// TIA Portal project "FactoryIO_Template_S7-1200_V15_V18" (V18)
// Vorlageprojekt für das Buch mit Zielsystem S7-1200

(* hardware
DEVICE "S7-1200-Station_1"  S7-1200 Station
   slot 0: "Baugruppenträger_0"  Rack  V1.0
   slot 1: "PLC_1"  CPU 1211C DC/DC/DC  6ES7 211-1AE40-0XB0  V4.1
DEVICE "HMI_1"  TP700 Comfort
   slot 0: "HMI_1"  TP700 Comfort  6AV2 124-0GC01-0AX0  17.0.0.0
   slot 1: "HMI_RT_1"  TP700 Comfort  6AV2 124-0GC01-0AX0  17.0.0.0
   slot 5: "HMI_1.IE_CP_1"  PROFINET Interface  17.0.0.0
      slot 1: "PROFINET Interface_1"  PROFINET Interface
         slot 1: "Port_1"  Port
         slot 2: "Port_2"  Port
   slot 7: "HMI_1.MPI/DP_CP_1"  MPI/DP Interface  17.0.0.0
DEVICE "PC station"  SIMATIC PC station
   slot 0: "PC station"  Rail  SIMATIC PC-Station  V1.0
      slot 125: "Stationmanager"  Station_Manager  V6.0.4
   slot 1: "IE general_1"  IE General  IE_CP  V8.2.0
      slot 1: "PROFINET interface"  IEGeneral.Interface.8.2.0
   slot 2: "HMI_RT_2"  WinCC RT Advanced  6AV2 104-0xxxx-xxxx  17.0.0.0
      slot 33792: "Computer interface"  Host interface
*)

// ===== PLC "PLC_1"  CPU 1211C DC/DC/DC =====

VAR_GLOBAL   // PLC tag table "Standard-Variablentabelle"
   "item at inter 0" AT %I0.0 : Bool;
   "item at exit 0" AT %I0.1 : Bool;
   "moving x0" AT %I0.2 : Bool;
   "moving z0" AT %I0.3 : Bool;
   "item detect 0" AT %I0.4 : Bool;
   "Start Button 0" AT %I0.5 : Bool;
   "Stop Button 0" AT %I0.6 : Bool;
   "Emergency Stop 0" AT %I0.7 : Bool;
   "enter conveyor (4m) 0" AT %Q0.0 : Bool;
   "exit conveyor (4m) 0" AT %Q0.1 : Bool;
   "move x0" AT %Q0.2 : Bool;
   "move z0" AT %Q0.3 : Bool;
   "grab 0" AT %Q0.4 : Bool;
   "Start Button 0 (Light)" AT %Q0.5 : Bool;
   "Stop Button 0 (Light)" AT %Q0.6 : Bool;
   "State0" AT %M1.0 : Bool;
   "State1" AT %M1.1 : Bool;
   "State2" AT %M1.2 : Bool;
   "State3" AT %M1.3 : Bool;
   "State4" AT %M1.4 : Bool;
   "State5" AT %M1.5 : Bool;
   "State6" AT %M1.6 : Bool;
   "State7" AT %M1.7 : Bool;
   "State8" AT %M2.0 : Bool;
   "State9" AT %M2.1 : Bool;
   "Tag_1" AT %M2.2 : Bool;
   "Tag_2" AT %M0.3 : Bool;
   "Tag_3" AT %M0.4 : Bool;
   "Tag_4" AT %M0.5 : Bool;
   "Tag_5" AT %M0.6 : Bool;
   "Tag_6" AT %M0.7 : Bool;
   "Digital Display 0" AT %QD30 : DInt;
   "Belt Conveyor (2m) 0" AT %Q0.7 : Bool;
   "Reset Button 0" AT %I1.0 : Bool;
   "Pusher 0" AT %Q1.0 : Bool;
   "Tag_7" AT %M0.0 : Bool;
   "Vision Sensor 3" AT %I1.1 : Bool;
   "Belt Conveyor (6m) 0" AT %Q1.1 : Bool;
   "Belt Conveyor (6m) 1" AT %Q1.2 : Bool;
   "Curved Belt Conveyor 0 CCW" AT %Q1.3 : Bool;
   "Curved Belt Conveyor 1 CW" AT %Q1.4 : Bool;
   "Belt Conveyor (6m) 2c1" AT %Q1.5 : Bool;
   "Belt Conveyor (6m) c_3_1" AT %Q1.6 : Bool;
   "Enter_sensor_green1" AT %I1.2 : Bool;
   "Exit_sensor_green" AT %I1.3 : Bool;
   "pusher_sensor" AT %I1.4 : Bool;
   "pusher_Sensor 2" AT %I1.5 : Bool;
   "Belt Conveyor (6m) 4" AT %Q1.7 : Bool;
   "Belt Conveyor (6m) 5" AT %Q2.0 : Bool;
   "Machining green(Start)" AT %Q2.1 : Bool;
   "Machining green  (Stop)" AT %Q2.2 : Bool;
   "Belt Conveyor (4m) 2c2" AT %Q2.3 : Bool;
   "Tag_8" AT %M2.3 : Bool;
   "reset_c1" AT %M2.4 : Bool;
   "Tag_9" AT %M2.5 : Bool;
   "Tag_10" AT %MW200 : Word;
   "reset_marker_lids" AT %M2.6 : Bool;
   "Tag_11" AT %M2.7 : Bool;
   "reset_c_1_b" AT %M3.0 : Bool;
   "Tag_12" AT %M3.1 : Bool;
   "reset_lib_blue" AT %M3.2 : Bool;
   "Tag_14" AT %MW300 : Int;
   "Tag_13" AT %M3.3 : Bool;
   "Tag_15" AT %M3.4 : Bool;
   "Tag_16" AT %M3.5 : Bool;
   "Tag_17" AT %M3.6 : Bool;
   "Tag_18" AT %M3.7 : Bool;
   "Tag_19" AT %M4.0 : Bool;
   "Tag_20" AT %M4.1 : Bool;
   "Tag_21" AT %M4.2 : Bool;
   "Tag_22" AT %M4.3 : Bool;
   "Tag_23" AT %M4.4 : Bool;
   "Tag_24" AT %M4.5 : Bool;
   "Tag_25" AT %M4.6 : Bool;
   "Tag_26" AT %M5.0 : Bool;
   "Tag_27" AT %M5.1 : Bool;
   "Tag_28" AT %M5.2 : Bool;
   "Tag_29" AT %M5.3 : Bool;
   "Tag_30" AT %M5.4 : Bool;
   "Tag_31" AT %MW400 : Int;
   "Tag_32" AT %M5.5 : Bool;
   "Tag_33" AT %MW500 : Int;
   "Tag_34" AT %MW600 : Int;
   "Tag_35" AT %M5.6 : Bool;
END_VAR

VAR_GLOBAL   // PLC tag table "Tag table from XML_1"
   "Digital Display 1" AT %QD34 : DInt;
   "Digital Display 2" AT %QD38 : DInt;
END_VAR

VAR_GLOBAL   // PLC tag table "Tag table from XML_4"
   "Enter_sensor_green2" AT %I1.6 : Bool;
END_VAR

VAR_GLOBAL   // PLC tag table "Tag table from XML_5"
   "Entry_sensor_blue_2_1" AT %I1.7 : Bool;
   "Entry_sensor_blue_2_2" AT %I2.0 : Bool;
   "Exit_sensor_blue_2" AT %I2.1 : Bool;
   "Start Button 1" AT %I2.2 : Bool;
   "Stop Button 1" AT %I2.3 : Bool;
   "Emergency Stop 1" AT %I2.4 : Bool;
   "Start Button 2" AT %I2.5 : Bool;
   "Stop Button 2" AT %I2.6 : Bool;
   "Emergency Stop 2" AT %I2.7 : Bool;
   "Start Button 3" AT %I3.0 : Bool;
   "Stop Button 3" AT %I3.1 : Bool;
   "Start Button 4" AT %I3.2 : Bool;
   "Stop Button 4" AT %I3.3 : Bool;
   "Moving X1" AT %I3.4 : Bool;
   "Moving Z1" AT %I3.5 : Bool;
   "Detected_item_1" AT %I3.6 : Bool;
   "Right Positioner 0 (Clamped)" AT %I3.7 : Bool;
   "Right Positioner 1 (Clamped)" AT %I4.0 : Bool;
   "Vision Sensor 0" AT %I4.1 : Bool;
   "Vision Sensor 1" AT %I4.2 : Bool;
   "push_sensor_2_1" AT %I4.3 : Bool;
   "push_sensor_2_2" AT %I4.4 : Bool;
   "push_sensor_3_1" AT %I4.5 : Bool;
   "push_sensor_3_2" AT %I4.6 : Bool;
   "counter_blue" AT %I4.7 : Bool;
   "counter_green" AT %I5.0 : Bool;
   "part_leveing1" AT %I5.1 : Bool;
   "part_leveing2" AT %I5.2 : Bool;
   "Moving X2" AT %I5.3 : Bool;
   "Moving Z2" AT %I5.4 : Bool;
   "Detected_item_2" AT %I5.5 : Bool;
   "Right Positioner 3 (Clamped)" AT %I5.6 : Bool;
   "Right Positioner 2 (Clamped)" AT %I5.7 : Bool;
   "Right Positioner 1 (Limit)" AT %I6.0 : Bool;
   "Right Positioner 3 (Limit)" AT %I6.1 : Bool;
   "Machining green lids" AT %Q2.4 : Bool;
   "Machining Center 0 (Produce Lids)" AT %Q2.5 : Bool;
   "Belt Conveyor (4m) c_3_2" AT %Q2.6 : Bool;
   "Start Button 1 (Light)" AT %Q2.7 : Bool;
   "Stop Button 1 (Light)" AT %Q3.0 : Bool;
   "Start Button 2 (Light)" AT %Q3.1 : Bool;
   "Stop Button 2 (Light)" AT %Q3.2 : Bool;
   "Start Button 3 (Light)" AT %Q3.3 : Bool;
   "Stop Button 3 (Light)" AT %Q3.4 : Bool;
   "Start Button 4 (Light)" AT %Q3.5 : Bool;
   "Stop Button 4 (Light)" AT %Q3.6 : Bool;
   "Curved Belt Conveyor 2 CCW" AT %Q3.7 : Bool;
   "Curved Belt Conveyor 3 CCW" AT %Q4.0 : Bool;
   "Belt Conveyor (4m) 3" AT %Q4.1 : Bool;
   "Belt Conveyor (4m) 4" AT %Q4.2 : Bool;
   "Belt Conveyor (4m) 5" AT %Q4.3 : Bool;
   "Belt Conveyor (4m) 6" AT %Q4.4 : Bool;
   "Move x1" AT %Q4.5 : Bool;
   "move z1" AT %Q4.6 : Bool;
   "Pusher _2" AT %Q4.7 : Bool;
   "Right Positioner 0 (Clamp)" AT %Q5.0 : Bool;
   "Right Positioner 1 (Clamp)" AT %Q5.1 : Bool;
   "Pusher_3" AT %Q5.2 : Bool;
   "Belt Conveyor (4m) 8" AT %Q5.3 : Bool;
   "Belt Conveyor (4m) 9" AT %Q5.4 : Bool;
   "Belt Conveyor (4m) 10" AT %Q5.5 : Bool;
   "Belt Conveyor (4m) 11" AT %Q5.6 : Bool;
   "move X2" AT %Q5.7 : Bool;
   "move z2" AT %Q6.0 : Bool;
   "Grab2" AT %Q6.1 : Bool;
   "Right Positioner 3 (Clamp)" AT %Q6.2 : Bool;
   "Right Positioner 2 (Clamp)" AT %Q6.3 : Bool;
   "Right Positioner 1 (Raise)" AT %Q6.4 : Bool;
   "Right Positioner 3 (Raise)" AT %Q6.5 : Bool;
END_VAR

VAR_GLOBAL   // PLC tag table "Tag table from XML_6"
   "Machining blue 0 (Start)" AT %Q6.6 : Bool;
   "Machining blue 0 (Stop)" AT %Q6.7 : Bool;
END_VAR

VAR_GLOBAL   // PLC tag table "Tag table from XML_7"
   "Grab1" AT %Q7.0 : Bool;
END_VAR

VAR_GLOBAL   // PLC tag table "Tag table from XML_8"
   "lid_place_blue" AT %I6.2 : Bool;
   "base_place_blue" AT %I6.3 : Bool;
   "lid_place_green" AT %I6.4 : Bool;
   "base_place_green" AT %I6.5 : Bool;
END_VAR

// folder: System blocks/Program resources

DATA_BLOCK "IEC_Counter_0_DB"   // DB1
{ S7_Optimized_Access := 'TRUE' }
AUTHOR : Simatic
FAMILY : IEC
NAME : CNTR
VERSION : 1.0
// stored: InstanceOfName IEC_COUNTER
"IEC_COUNTER"
BEGIN
END_DATA_BLOCK

DATA_BLOCK "IEC_Timer_0_DB"   // DB2
{ S7_Optimized_Access := 'TRUE' }
AUTHOR : Simatic
FAMILY : IEC
NAME : IEC_TMR
VERSION : 1.0
// stored: InstanceOfName IEC_TIMER
"IEC_TIMER"
BEGIN
END_DATA_BLOCK

DATA_BLOCK "IEC_Timer_0_DB_1"   // DB3
{ S7_Optimized_Access := 'TRUE' }
AUTHOR : Simatic
FAMILY : IEC
NAME : IEC_TMR
VERSION : 1.0
// stored: InstanceOfName IEC_TIMER
"IEC_TIMER"
BEGIN
END_DATA_BLOCK

DATA_BLOCK "produce_lids_counter"   // DB4
{ S7_Optimized_Access := 'TRUE' }
AUTHOR : Simatic
FAMILY : IEC
NAME : CNTR
VERSION : 1.0
// stored: InstanceOfName IEC_COUNTER
"IEC_COUNTER"
BEGIN
END_DATA_BLOCK

DATA_BLOCK "IEC_Timer_0_DB_2"   // DB5
{ S7_Optimized_Access := 'TRUE' }
AUTHOR : Simatic
FAMILY : IEC
NAME : IEC_TMR
VERSION : 1.0
// stored: InstanceOfName IEC_TIMER
"IEC_TIMER"
BEGIN
END_DATA_BLOCK

DATA_BLOCK "IEC_Timer_0_DB_3"   // DB6
{ S7_Optimized_Access := 'TRUE' }
AUTHOR : Simatic
FAMILY : IEC
NAME : IEC_TMR
VERSION : 1.0
// stored: InstanceOfName IEC_TIMER
"IEC_TIMER"
BEGIN
END_DATA_BLOCK

DATA_BLOCK "produce_lids_counter_blue"   // DB7
{ S7_Optimized_Access := 'TRUE' }
AUTHOR : Simatic
FAMILY : IEC
NAME : CNTR
VERSION : 1.0
// stored: InstanceOfName IEC_COUNTER
"IEC_COUNTER"
BEGIN
END_DATA_BLOCK

DATA_BLOCK "Green_Product_Counter"   // DB9
{ S7_Optimized_Access := 'TRUE' }
AUTHOR : Simatic
FAMILY : IEC
NAME : CNTR
VERSION : 1.0
// stored: InstanceOfName IEC_COUNTER
"IEC_COUNTER"
BEGIN
END_DATA_BLOCK

DATA_BLOCK "Blue_Product_Counter"   // DB10
{ S7_Optimized_Access := 'TRUE' }
AUTHOR : Simatic
FAMILY : IEC
NAME : CNTR
VERSION : 1.0
// stored: InstanceOfName IEC_COUNTER
"IEC_COUNTER"
BEGIN
END_DATA_BLOCK

// folder: (top level)

FUNCTION "Start_Stop" : Void   // FC1, LAD
{ S7_Optimized_Access := 'TRUE' }
VERSION : 0.1
BEGIN

REGION Network 1
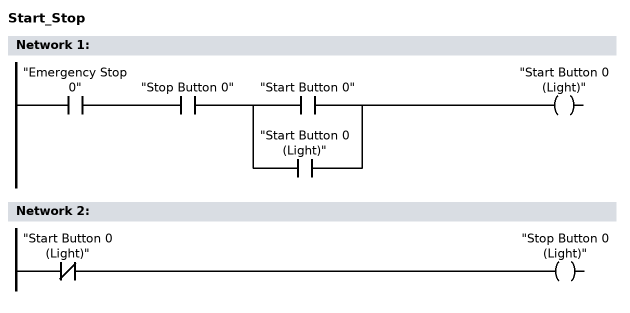
   RUNG wire#powerrail
      Contact( "Emergency Stop 0" )
      Contact( "Stop Button 0" )
      wire#w1
      Contact( "Start Button 0" )
      wire#w2
      Coil( "Start Button 0 (Light)" )
   END_RUNG
   RUNG wire#w1
      Contact( "Start Button 0 (Light)" )
   END_RUNG wire#w2
   // the same network as SCL:
   "Start Button 0 (Light)" := "Emergency Stop 0" AND "Stop Button 0" AND ("Start Button 0" OR "Start Button 0 (Light)");
END_REGION

REGION Network 2
   RUNG wire#powerrail
      I_Contact( "Start Button 0 (Light)" )
      Coil( "Stop Button 0 (Light)" )
   END_RUNG
   // the same network as SCL:
   "Stop Button 0 (Light)" := NOT "Start Button 0 (Light)";
END_REGION
END_FUNCTION

FUNCTION "States" : Void   // FC2, LAD
{ S7_Optimized_Access := 'TRUE' }
VERSION : 0.1
   VAR_TEMP   // added for the SCL form of the ladder/FBD networks
      _w1 : Bool;
   END_VAR
BEGIN

REGION Network 1: State0
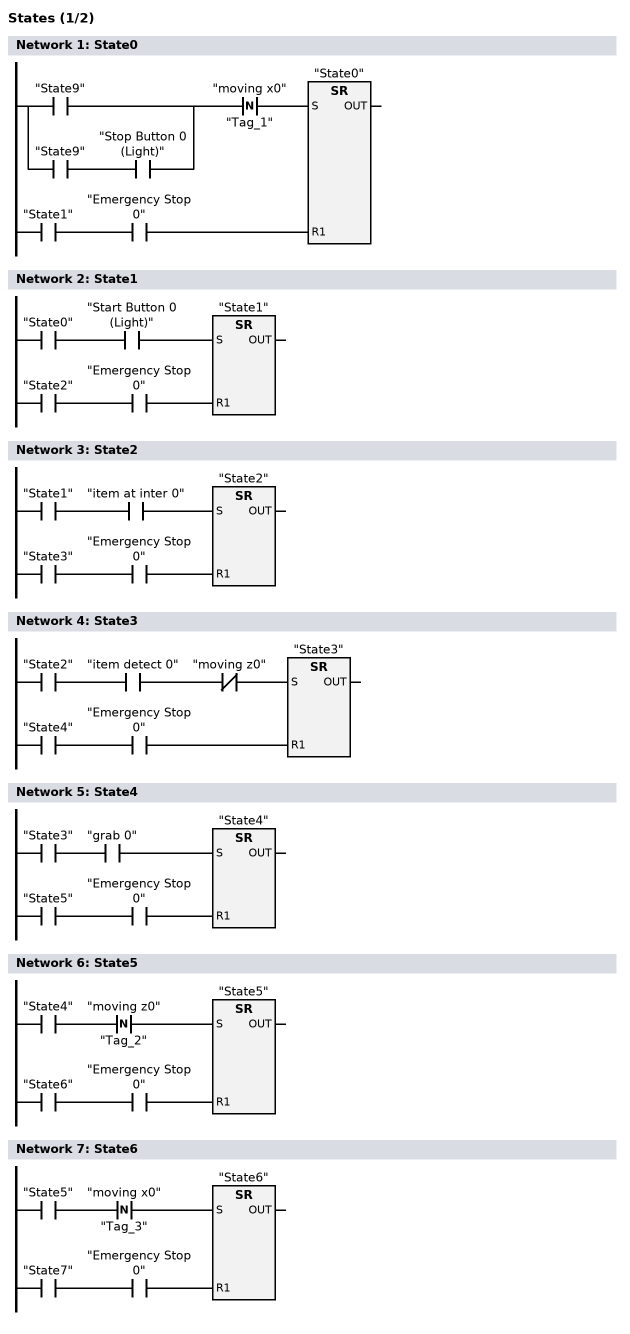
   RUNG wire#powerrail
      Contact( "State9" )
      wire#w1
      N_Contact(operand := "moving x0", bit := "Tag_1")
      S_SR(operand := "State0", r1 := wire#w2)
   END_RUNG
   RUNG wire#powerrail
      Contact( "State9" )
      Contact( "Stop Button 0 (Light)" )
   END_RUNG wire#w1
   RUNG wire#powerrail
      Contact( "State1" )
      Contact( "Emergency Stop 0" )
   END_RUNG wire#w2
   // the same network as SCL:
   #_w1 := ("State9" OR ("State9" AND "Stop Button 0 (Light)")) AND NOT "moving x0" AND "Tag_1";   // falling edge of "moving x0"
   "Tag_1" := "moving x0";
   IF #_w1 THEN
       "State0" := TRUE;   // SR flip-flop
   END_IF;
   IF "State1" AND "Emergency Stop 0" THEN "State0" := FALSE; END_IF;
END_REGION

REGION Network 2: State1
   RUNG wire#powerrail
      Contact( "State0" )
      Contact( "Start Button 0 (Light)" )
      S_SR(operand := "State1", r1 := wire#w1)
   END_RUNG
   RUNG wire#powerrail
      Contact( "State2" )
      Contact( "Emergency Stop 0" )
   END_RUNG wire#w1
   // the same network as SCL:
   IF "State0" AND "Start Button 0 (Light)" THEN
       "State1" := TRUE;   // SR flip-flop
   END_IF;
   IF "State2" AND "Emergency Stop 0" THEN "State1" := FALSE; END_IF;
END_REGION

REGION Network 3: State2
   RUNG wire#powerrail
      Contact( "State1" )
      Contact( "item at inter 0" )
      S_SR(operand := "State2", r1 := wire#w1)
   END_RUNG
   RUNG wire#powerrail
      Contact( "State3" )
      Contact( "Emergency Stop 0" )
   END_RUNG wire#w1
   // the same network as SCL:
   IF "State1" AND "item at inter 0" THEN
       "State2" := TRUE;   // SR flip-flop
   END_IF;
   IF "State3" AND "Emergency Stop 0" THEN "State2" := FALSE; END_IF;
END_REGION

REGION Network 4: State3
   RUNG wire#powerrail
      Contact( "State2" )
      Contact( "item detect 0" )
      I_Contact( "moving z0" )
      S_SR(operand := "State3", r1 := wire#w1)
   END_RUNG
   RUNG wire#powerrail
      Contact( "State4" )
      Contact( "Emergency Stop 0" )
   END_RUNG wire#w1
   // the same network as SCL:
   IF "State2" AND "item detect 0" AND NOT "moving z0" THEN
       "State3" := TRUE;   // SR flip-flop
   END_IF;
   IF "State4" AND "Emergency Stop 0" THEN "State3" := FALSE; END_IF;
END_REGION

REGION Network 5: State4
   RUNG wire#powerrail
      Contact( "State3" )
      Contact( "grab 0" )
      S_SR(operand := "State4", r1 := wire#w1)
   END_RUNG
   RUNG wire#powerrail
      Contact( "State5" )
      Contact( "Emergency Stop 0" )
   END_RUNG wire#w1
   // the same network as SCL:
   IF "State3" AND "grab 0" THEN
       "State4" := TRUE;   // SR flip-flop
   END_IF;
   IF "State5" AND "Emergency Stop 0" THEN "State4" := FALSE; END_IF;
END_REGION

REGION Network 6: State5
   RUNG wire#powerrail
      Contact( "State4" )
      N_Contact(operand := "moving z0", bit := "Tag_2")
      S_SR(operand := "State5", r1 := wire#w1)
   END_RUNG
   RUNG wire#powerrail
      Contact( "State6" )
      Contact( "Emergency Stop 0" )
   END_RUNG wire#w1
   // the same network as SCL:
   #_w1 := "State4" AND NOT "moving z0" AND "Tag_2";   // falling edge of "moving z0"
   "Tag_2" := "moving z0";
   IF #_w1 THEN
       "State5" := TRUE;   // SR flip-flop
   END_IF;
   IF "State6" AND "Emergency Stop 0" THEN "State5" := FALSE; END_IF;
END_REGION

REGION Network 7: State6
   RUNG wire#powerrail
      Contact( "State5" )
      N_Contact(operand := "moving x0", bit := "Tag_3")
      S_SR(operand := "State6", r1 := wire#w1)
   END_RUNG
   RUNG wire#powerrail
      Contact( "State7" )
      Contact( "Emergency Stop 0" )
   END_RUNG wire#w1
   // the same network as SCL:
   #_w1 := "State5" AND NOT "moving x0" AND "Tag_3";   // falling edge of "moving x0"
   "Tag_3" := "moving x0";
   IF #_w1 THEN
       "State6" := TRUE;   // SR flip-flop
   END_IF;
   IF "State7" AND "Emergency Stop 0" THEN "State6" := FALSE; END_IF;
END_REGION

REGION Network 8: State7
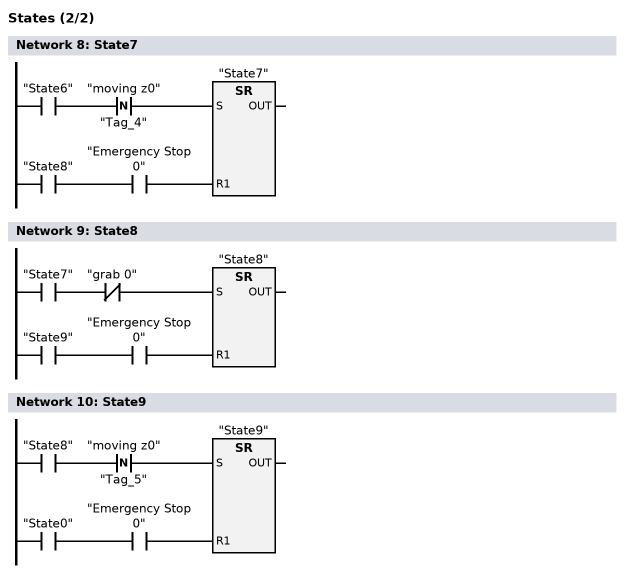
   RUNG wire#powerrail
      Contact( "State6" )
      N_Contact(operand := "moving z0", bit := "Tag_4")
      S_SR(operand := "State7", r1 := wire#w1)
   END_RUNG
   RUNG wire#powerrail
      Contact( "State8" )
      Contact( "Emergency Stop 0" )
   END_RUNG wire#w1
   // the same network as SCL:
   #_w1 := "State6" AND NOT "moving z0" AND "Tag_4";   // falling edge of "moving z0"
   "Tag_4" := "moving z0";
   IF #_w1 THEN
       "State7" := TRUE;   // SR flip-flop
   END_IF;
   IF "State8" AND "Emergency Stop 0" THEN "State7" := FALSE; END_IF;
END_REGION

REGION Network 9: State8
   RUNG wire#powerrail
      Contact( "State7" )
      I_Contact( "grab 0" )
      S_SR(operand := "State8", r1 := wire#w1)
   END_RUNG
   RUNG wire#powerrail
      Contact( "State9" )
      Contact( "Emergency Stop 0" )
   END_RUNG wire#w1
   // the same network as SCL:
   IF "State7" AND NOT "grab 0" THEN
       "State8" := TRUE;   // SR flip-flop
   END_IF;
   IF "State9" AND "Emergency Stop 0" THEN "State8" := FALSE; END_IF;
END_REGION

REGION Network 10: State9
   RUNG wire#powerrail
      Contact( "State8" )
      N_Contact(operand := "moving z0", bit := "Tag_5")
      S_SR(operand := "State9", r1 := wire#w1)
   END_RUNG
   RUNG wire#powerrail
      Contact( "State0" )
      Contact( "Emergency Stop 0" )
   END_RUNG wire#w1
   // the same network as SCL:
   #_w1 := "State8" AND NOT "moving z0" AND "Tag_5";   // falling edge of "moving z0"
   "Tag_5" := "moving z0";
   IF #_w1 THEN
       "State9" := TRUE;   // SR flip-flop
   END_IF;
   IF "State0" AND "Emergency Stop 0" THEN "State9" := FALSE; END_IF;
END_REGION
END_FUNCTION

FUNCTION "Actuators" : Void   // FC3, LAD
{ S7_Optimized_Access := 'TRUE' }
VERSION : 0.1
BEGIN

REGION Network 1
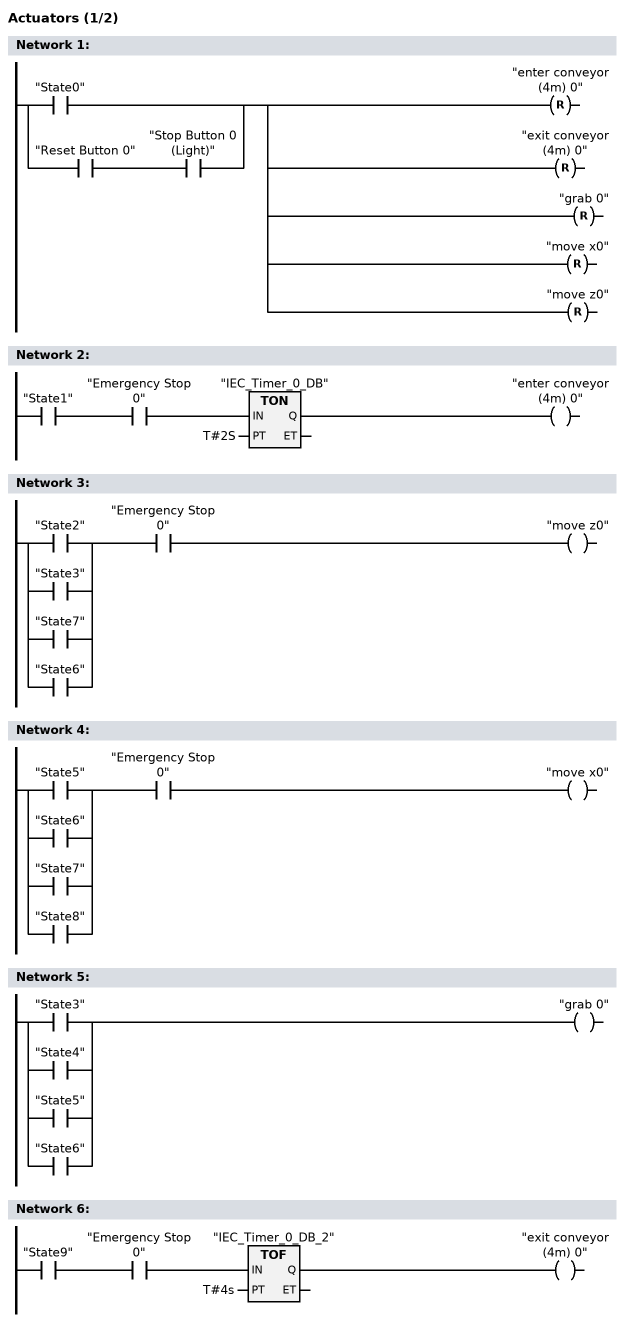
   RUNG wire#powerrail
      Contact( "State0" )
      wire#w1
      R_Coil( "enter conveyor (4m) 0" )
   END_RUNG
   RUNG wire#powerrail
      Contact( "Reset Button 0" )
      Contact( "Stop Button 0 (Light)" )
   END_RUNG wire#w1
   RUNG wire#w1
      R_Coil( "exit conveyor (4m) 0" )
   END_RUNG
   RUNG wire#w1
      R_Coil( "grab 0" )
   END_RUNG
   RUNG wire#w1
      R_Coil( "move x0" )
   END_RUNG
   RUNG wire#w1
      R_Coil( "move z0" )
   END_RUNG
   // the same network as SCL:
   IF "State0" OR ("Reset Button 0" AND "Stop Button 0 (Light)") THEN
       "enter conveyor (4m) 0" := FALSE;
       "exit conveyor (4m) 0" := FALSE;
       "grab 0" := FALSE;
       "move x0" := FALSE;
       "move z0" := FALSE;
   END_IF;
END_REGION

REGION Network 2
   "IEC_Timer_0_DB".TON(IN := "State1" AND "Emergency Stop 0", PT := T#2S);
   "enter conveyor (4m) 0" := "IEC_Timer_0_DB".Q;
END_REGION

REGION Network 3
   RUNG wire#powerrail
      Contact( "State2" )
      wire#w1
      Contact( "Emergency Stop 0" )
      Coil( "move z0" )
   END_RUNG
   RUNG wire#powerrail
      Contact( "State3" )
   END_RUNG wire#w1
   RUNG wire#powerrail
      Contact( "State7" )
   END_RUNG wire#w1
   RUNG wire#powerrail
      Contact( "State6" )
   END_RUNG wire#w1
   // the same network as SCL:
   "move z0" := ("State2" OR "State3" OR "State7" OR "State6") AND "Emergency Stop 0";
END_REGION

REGION Network 4
   RUNG wire#powerrail
      Contact( "State5" )
      wire#w1
      Contact( "Emergency Stop 0" )
      Coil( "move x0" )
   END_RUNG
   RUNG wire#powerrail
      Contact( "State6" )
   END_RUNG wire#w1
   RUNG wire#powerrail
      Contact( "State7" )
   END_RUNG wire#w1
   RUNG wire#powerrail
      Contact( "State8" )
   END_RUNG wire#w1
   // the same network as SCL:
   "move x0" := ("State5" OR "State6" OR "State7" OR "State8") AND "Emergency Stop 0";
END_REGION

REGION Network 5
   RUNG wire#powerrail
      Contact( "State3" )
      wire#w1
      Coil( "grab 0" )
   END_RUNG
   RUNG wire#powerrail
      Contact( "State4" )
   END_RUNG wire#w1
   RUNG wire#powerrail
      Contact( "State5" )
   END_RUNG wire#w1
   RUNG wire#powerrail
      Contact( "State6" )
   END_RUNG wire#w1
   // the same network as SCL:
   "grab 0" := "State3" OR "State4" OR "State5" OR "State6";
END_REGION

REGION Network 6
   "IEC_Timer_0_DB_2".TOF(IN := "State9" AND "Emergency Stop 0", PT := T#4s);
   "exit conveyor (4m) 0" := "IEC_Timer_0_DB_2".Q;
END_REGION

REGION Network 7
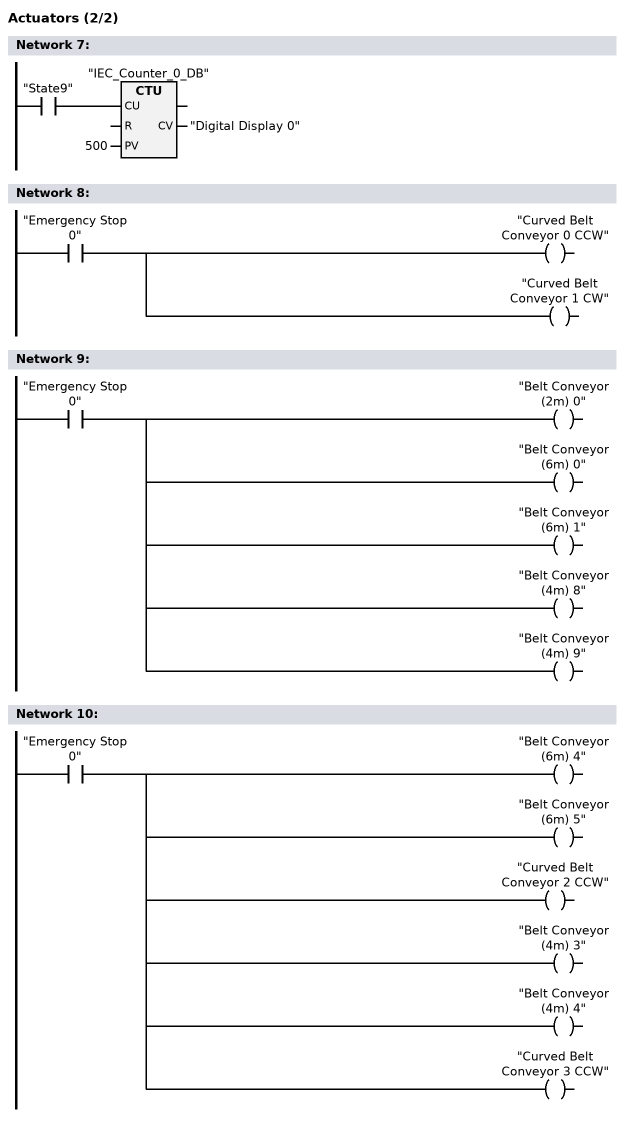
   "IEC_Counter_0_DB".CTU(CU := "State9", PV := 500, CV => "Digital Display 0");
END_REGION

REGION Network 8
   RUNG wire#powerrail
      Contact( "Emergency Stop 0" )
      wire#w1
      Coil( "Curved Belt Conveyor 0 CCW" )
   END_RUNG
   RUNG wire#w1
      Coil( "Curved Belt Conveyor 1 CW" )
   END_RUNG
   // the same network as SCL:
   "Curved Belt Conveyor 0 CCW" := "Emergency Stop 0";
   "Curved Belt Conveyor 1 CW" := "Emergency Stop 0";
END_REGION

REGION Network 9
   RUNG wire#powerrail
      Contact( "Emergency Stop 0" )
      wire#w1
      Coil( "Belt Conveyor (2m) 0" )
   END_RUNG
   RUNG wire#w1
      Coil( "Belt Conveyor (6m) 0" )
   END_RUNG
   RUNG wire#w1
      Coil( "Belt Conveyor (6m) 1" )
   END_RUNG
   RUNG wire#w1
      Coil( "Belt Conveyor (4m) 8" )
   END_RUNG
   RUNG wire#w1
      Coil( "Belt Conveyor (4m) 9" )
   END_RUNG
   // the same network as SCL:
   "Belt Conveyor (2m) 0" := "Emergency Stop 0";
   "Belt Conveyor (6m) 0" := "Emergency Stop 0";
   "Belt Conveyor (6m) 1" := "Emergency Stop 0";
   "Belt Conveyor (4m) 8" := "Emergency Stop 0";
   "Belt Conveyor (4m) 9" := "Emergency Stop 0";
END_REGION

REGION Network 10
   RUNG wire#powerrail
      Contact( "Emergency Stop 0" )
      wire#w1
      Coil( "Belt Conveyor (6m) 4" )
   END_RUNG
   RUNG wire#w1
      Coil( "Belt Conveyor (6m) 5" )
   END_RUNG
   RUNG wire#w1
      Coil( "Curved Belt Conveyor 2 CCW" )
   END_RUNG
   RUNG wire#w1
      Coil( "Belt Conveyor (4m) 3" )
   END_RUNG
   RUNG wire#w1
      Coil( "Belt Conveyor (4m) 4" )
   END_RUNG
   RUNG wire#w1
      Coil( "Curved Belt Conveyor 3 CCW" )
   END_RUNG
   // the same network as SCL:
   "Belt Conveyor (6m) 4" := "Emergency Stop 0";
   "Belt Conveyor (6m) 5" := "Emergency Stop 0";
   "Curved Belt Conveyor 2 CCW" := "Emergency Stop 0";
   "Belt Conveyor (4m) 3" := "Emergency Stop 0";
   "Belt Conveyor (4m) 4" := "Emergency Stop 0";
   "Curved Belt Conveyor 3 CCW" := "Emergency Stop 0";
END_REGION
END_FUNCTION

FUNCTION "CNC_BLUE" : Void   // FC4, LAD
{ S7_Optimized_Access := 'TRUE' }
VERSION : 0.1
BEGIN

REGION Network 1
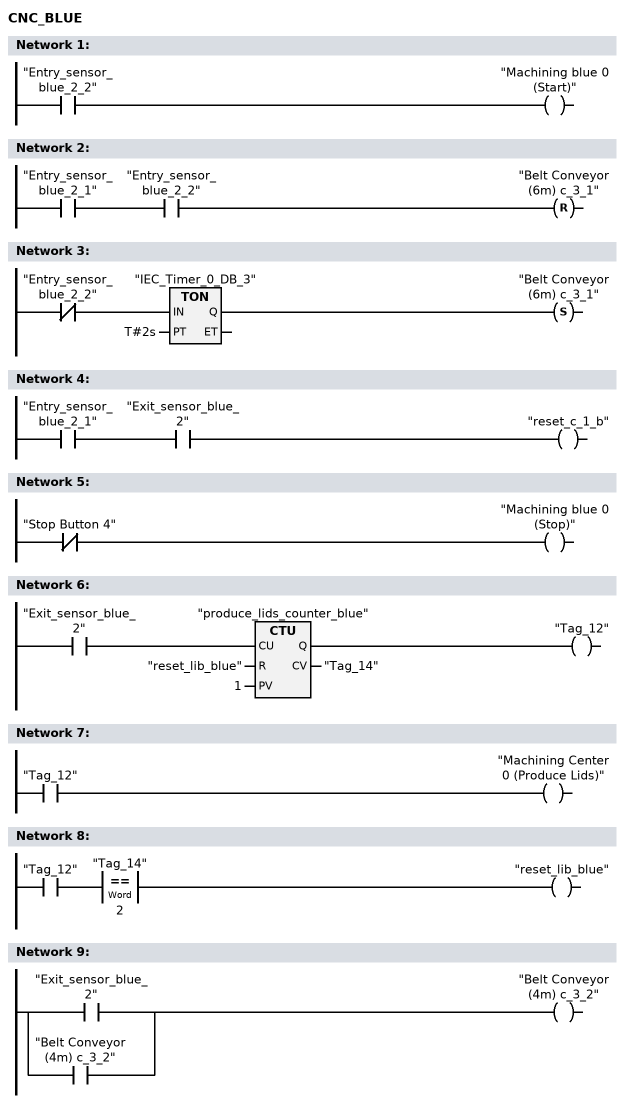
   RUNG wire#powerrail
      Contact( "Entry_sensor_blue_2_2" )
      Coil( "Machining blue 0 (Start)" )
   END_RUNG
   // the same network as SCL:
   "Machining blue 0 (Start)" := "Entry_sensor_blue_2_2";
END_REGION

REGION Network 2
   RUNG wire#powerrail
      Contact( "Entry_sensor_blue_2_1" )
      Contact( "Entry_sensor_blue_2_2" )
      R_Coil( "Belt Conveyor (6m) c_3_1" )
   END_RUNG
   // the same network as SCL:
   IF "Entry_sensor_blue_2_1" AND "Entry_sensor_blue_2_2" THEN "Belt Conveyor (6m) c_3_1" := FALSE; END_IF;
END_REGION

REGION Network 3
   "IEC_Timer_0_DB_3".TON(IN := NOT "Entry_sensor_blue_2_2", PT := T#2s);
   IF "IEC_Timer_0_DB_3".Q THEN "Belt Conveyor (6m) c_3_1" := TRUE; END_IF;
END_REGION

REGION Network 4
   RUNG wire#powerrail
      Contact( "Entry_sensor_blue_2_1" )
      Contact( "Exit_sensor_blue_2" )
      Coil( "reset_c_1_b" )
   END_RUNG
   // the same network as SCL:
   "reset_c_1_b" := "Entry_sensor_blue_2_1" AND "Exit_sensor_blue_2";
END_REGION

REGION Network 5
   RUNG wire#powerrail
      I_Contact( "Stop Button 4" )
      Coil( "Machining blue 0 (Stop)" )
   END_RUNG
   // the same network as SCL:
   "Machining blue 0 (Stop)" := NOT "Stop Button 4";
END_REGION

REGION Network 6
   "produce_lids_counter_blue".CTU(CU := "Exit_sensor_blue_2", R := "reset_lib_blue", PV := 1, CV => "Tag_14");
   "Tag_12" := "produce_lids_counter_blue".Q;
END_REGION

REGION Network 7
   RUNG wire#powerrail
      Contact( "Tag_12" )
      Coil( "Machining Center 0 (Produce Lids)" )
   END_RUNG
   // the same network as SCL:
   "Machining Center 0 (Produce Lids)" := "Tag_12";
END_REGION

REGION Network 8
   RUNG wire#powerrail
      Contact( "Tag_12" )
      { S7_Templates := "SrcType := Word" } EQ_Contact(in1 := "Tag_14", in2 := 2)
      Coil( "reset_lib_blue" )
   END_RUNG
   // the same network as SCL:
   "reset_lib_blue" := "Tag_12" AND ("Tag_14" = 2);
END_REGION

REGION Network 9
   RUNG wire#powerrail
      Contact( "Exit_sensor_blue_2" )
      wire#w1
      Coil( "Belt Conveyor (4m) c_3_2" )
   END_RUNG
   RUNG wire#powerrail
      Contact( "Belt Conveyor (4m) c_3_2" )
   END_RUNG wire#w1
   // the same network as SCL:
   "Belt Conveyor (4m) c_3_2" := "Exit_sensor_blue_2" OR "Belt Conveyor (4m) c_3_2";
END_REGION
END_FUNCTION

FUNCTION "CNC_GREEN" : Void   // FC5, LAD
{ S7_Optimized_Access := 'TRUE' }
VERSION : 0.1
BEGIN

REGION Network 1
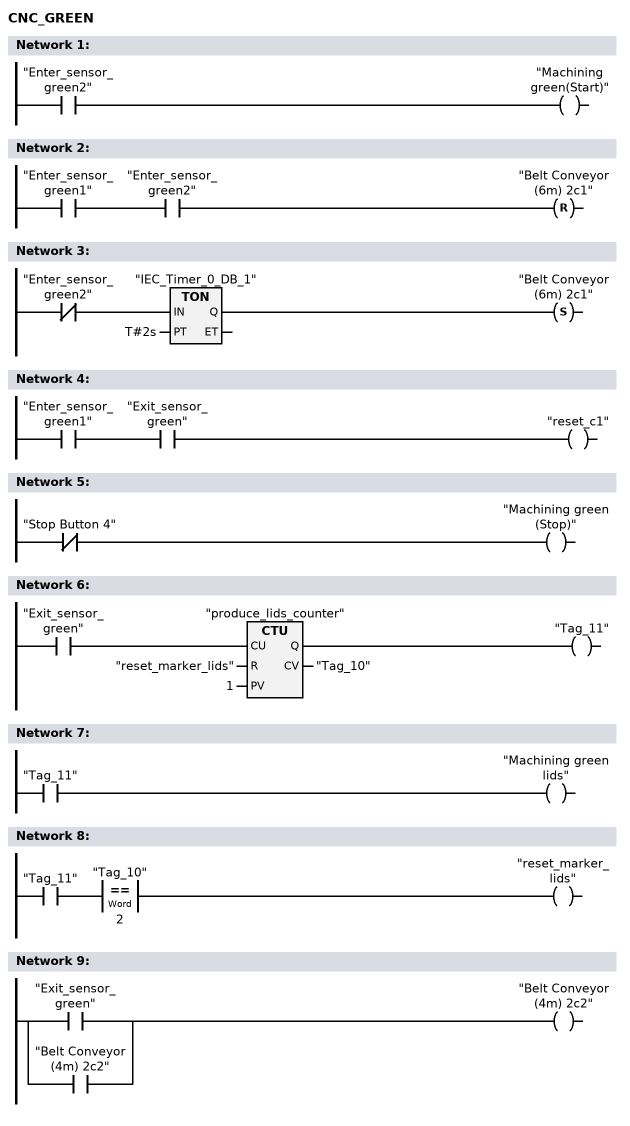
   RUNG wire#powerrail
      Contact( "Enter_sensor_green2" )
      Coil( "Machining green(Start)" )
   END_RUNG
   // the same network as SCL:
   "Machining green(Start)" := "Enter_sensor_green2";
END_REGION

REGION Network 2
   RUNG wire#powerrail
      Contact( "Enter_sensor_green1" )
      Contact( "Enter_sensor_green2" )
      R_Coil( "Belt Conveyor (6m) 2c1" )
   END_RUNG
   // the same network as SCL:
   IF "Enter_sensor_green1" AND "Enter_sensor_green2" THEN "Belt Conveyor (6m) 2c1" := FALSE; END_IF;
END_REGION

REGION Network 3
   "IEC_Timer_0_DB_1".TON(IN := NOT "Enter_sensor_green2", PT := T#2s);
   IF "IEC_Timer_0_DB_1".Q THEN "Belt Conveyor (6m) 2c1" := TRUE; END_IF;
END_REGION

REGION Network 4
   RUNG wire#powerrail
      Contact( "Enter_sensor_green1" )
      Contact( "Exit_sensor_green" )
      Coil( "reset_c1" )
   END_RUNG
   // the same network as SCL:
   "reset_c1" := "Enter_sensor_green1" AND "Exit_sensor_green";
END_REGION

REGION Network 5
   RUNG wire#powerrail
      I_Contact( "Stop Button 4" )
      Coil( "Machining green  (Stop)" )
   END_RUNG
   // the same network as SCL:
   "Machining green  (Stop)" := NOT "Stop Button 4";
END_REGION

REGION Network 6
   "produce_lids_counter".CTU(CU := "Exit_sensor_green", R := "reset_marker_lids", PV := 1, CV => "Tag_10");
   "Tag_11" := "produce_lids_counter".Q;
END_REGION

REGION Network 7
   RUNG wire#powerrail
      Contact( "Tag_11" )
      Coil( "Machining green lids" )
   END_RUNG
   // the same network as SCL:
   "Machining green lids" := "Tag_11";
END_REGION

REGION Network 8
   RUNG wire#powerrail
      Contact( "Tag_11" )
      { S7_Templates := "SrcType := Word" } EQ_Contact(in1 := "Tag_10", in2 := 2)
      Coil( "reset_marker_lids" )
   END_RUNG
   // the same network as SCL:
   "reset_marker_lids" := "Tag_11" AND ("Tag_10" = 2);
END_REGION

REGION Network 9
   RUNG wire#powerrail
      Contact( "Exit_sensor_green" )
      wire#w1
      Coil( "Belt Conveyor (4m) 2c2" )
   END_RUNG
   RUNG wire#powerrail
      Contact( "Belt Conveyor (4m) 2c2" )
   END_RUNG wire#w1
   // the same network as SCL:
   "Belt Conveyor (4m) 2c2" := "Exit_sensor_green" OR "Belt Conveyor (4m) 2c2";
END_REGION
END_FUNCTION

FUNCTION "Sorting" : Void   // FC6, LAD
{ S7_Optimized_Access := 'TRUE' }
VERSION : 0.1
BEGIN

REGION Network 1
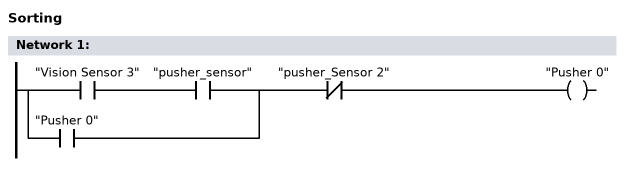
   RUNG wire#powerrail
      Contact( "Vision Sensor 3" )
      Contact( "pusher_sensor" )
      wire#w1
      I_Contact( "pusher_Sensor 2" )
      Coil( "Pusher 0" )
   END_RUNG
   RUNG wire#powerrail
      Contact( "Pusher 0" )
   END_RUNG wire#w1
   // the same network as SCL:
   "Pusher 0" := (("Vision Sensor 3" AND "pusher_sensor") OR "Pusher 0") AND NOT "pusher_Sensor 2";
END_REGION
END_FUNCTION

FUNCTION "Assimply_green" : Void   // FC7, LAD
{ S7_Optimized_Access := 'TRUE' }
VERSION : 0.1
   VAR_TEMP   // added for the SCL form of the ladder/FBD networks
      _w1 : Bool;
      _w2 : Bool;
   END_VAR
BEGIN

REGION Network 1
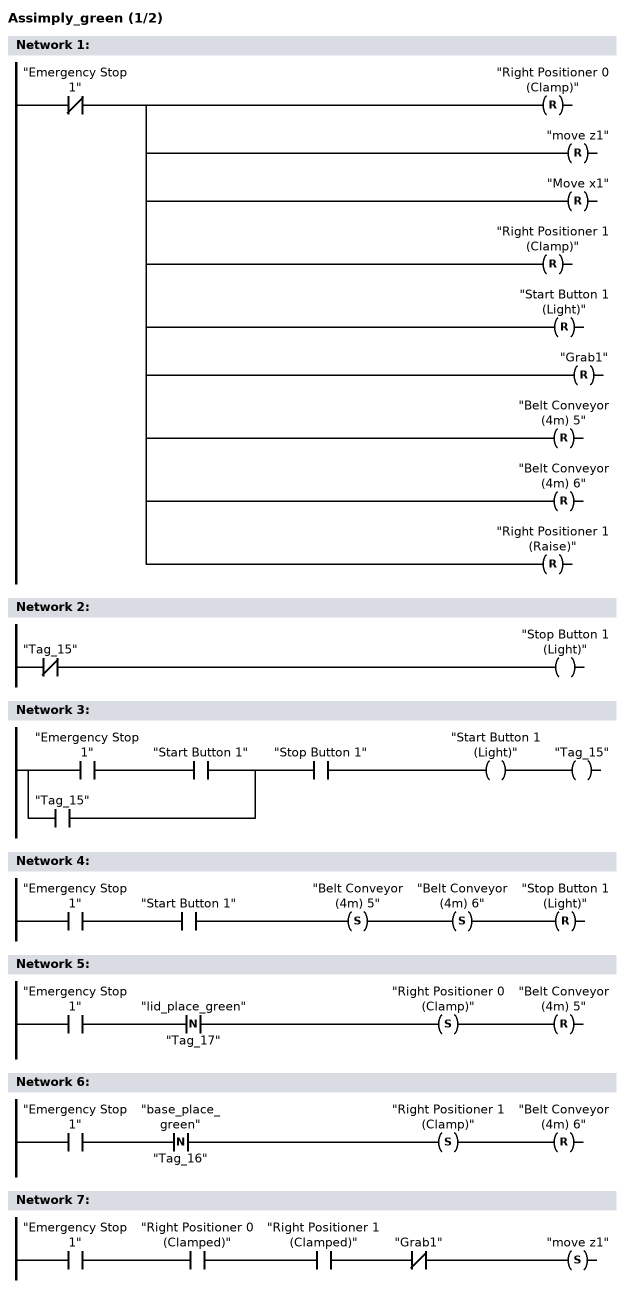
   RUNG wire#powerrail
      I_Contact( "Emergency Stop 1" )
      wire#w1
      R_Coil( "Right Positioner 0 (Clamp)" )
   END_RUNG
   RUNG wire#w1
      R_Coil( "move z1" )
   END_RUNG
   RUNG wire#w1
      R_Coil( "Move x1" )
   END_RUNG
   RUNG wire#w1
      R_Coil( "Right Positioner 1 (Clamp)" )
   END_RUNG
   RUNG wire#w1
      R_Coil( "Start Button 1 (Light)" )
   END_RUNG
   RUNG wire#w1
      R_Coil( "Grab1" )
   END_RUNG
   RUNG wire#w1
      R_Coil( "Belt Conveyor (4m) 5" )
   END_RUNG
   RUNG wire#w1
      R_Coil( "Belt Conveyor (4m) 6" )
   END_RUNG
   RUNG wire#w1
      R_Coil( "Right Positioner 1 (Raise)" )
   END_RUNG
   // the same network as SCL:
   IF NOT "Emergency Stop 1" THEN
       "Right Positioner 0 (Clamp)" := FALSE;
       "move z1" := FALSE;
       "Move x1" := FALSE;
       "Right Positioner 1 (Clamp)" := FALSE;
       "Start Button 1 (Light)" := FALSE;
       "Grab1" := FALSE;
       "Belt Conveyor (4m) 5" := FALSE;
       "Belt Conveyor (4m) 6" := FALSE;
       "Right Positioner 1 (Raise)" := FALSE;
   END_IF;
END_REGION

REGION Network 2
   RUNG wire#powerrail
      I_Contact( "Tag_15" )
      Coil( "Stop Button 1 (Light)" )
   END_RUNG
   // the same network as SCL:
   "Stop Button 1 (Light)" := NOT "Tag_15";
END_REGION

REGION Network 3
   RUNG wire#powerrail
      Contact( "Emergency Stop 1" )
      Contact( "Start Button 1" )
      wire#w1
      Contact( "Stop Button 1" )
      Coil( "Start Button 1 (Light)" )
      Coil( "Tag_15" )
   END_RUNG
   RUNG wire#powerrail
      Contact( "Tag_15" )
   END_RUNG wire#w1
   // the same network as SCL:
   "Start Button 1 (Light)" := (("Emergency Stop 1" AND "Start Button 1") OR "Tag_15") AND "Stop Button 1";
   "Tag_15" := "Start Button 1 (Light)";
END_REGION

REGION Network 4
   RUNG wire#powerrail
      Contact( "Emergency Stop 1" )
      Contact( "Start Button 1" )
      S_Coil( "Belt Conveyor (4m) 5" )
      S_Coil( "Belt Conveyor (4m) 6" )
      R_Coil( "Stop Button 1 (Light)" )
   END_RUNG
   // the same network as SCL:
   IF "Emergency Stop 1" AND "Start Button 1" THEN
       "Belt Conveyor (4m) 5" := TRUE;
       "Belt Conveyor (4m) 6" := TRUE;
       "Stop Button 1 (Light)" := FALSE;
   END_IF;
END_REGION

REGION Network 5
   RUNG wire#powerrail
      Contact( "Emergency Stop 1" )
      N_Contact(operand := "lid_place_green", bit := "Tag_17")
      S_Coil( "Right Positioner 0 (Clamp)" )
      R_Coil( "Belt Conveyor (4m) 5" )
   END_RUNG
   // the same network as SCL:
   #_w1 := "Emergency Stop 1" AND NOT "lid_place_green" AND "Tag_17";   // falling edge of "lid_place_green"
   "Tag_17" := "lid_place_green";
   IF #_w1 THEN
       "Right Positioner 0 (Clamp)" := TRUE;
       "Belt Conveyor (4m) 5" := FALSE;
   END_IF;
END_REGION

REGION Network 6
   RUNG wire#powerrail
      Contact( "Emergency Stop 1" )
      N_Contact(operand := "base_place_green", bit := "Tag_16")
      S_Coil( "Right Positioner 1 (Clamp)" )
      R_Coil( "Belt Conveyor (4m) 6" )
   END_RUNG
   // the same network as SCL:
   #_w1 := "Emergency Stop 1" AND NOT "base_place_green" AND "Tag_16";   // falling edge of "base_place_green"
   "Tag_16" := "base_place_green";
   IF #_w1 THEN
       "Right Positioner 1 (Clamp)" := TRUE;
       "Belt Conveyor (4m) 6" := FALSE;
   END_IF;
END_REGION

REGION Network 7
   RUNG wire#powerrail
      Contact( "Emergency Stop 1" )
      Contact( "Right Positioner 0 (Clamped)" )
      Contact( "Right Positioner 1 (Clamped)" )
      I_Contact( "Grab1" )
      S_Coil( "move z1" )
   END_RUNG
   // the same network as SCL:
   IF "Emergency Stop 1" AND "Right Positioner 0 (Clamped)" AND "Right Positioner 1 (Clamped)" AND NOT "Grab1" THEN
       "move z1" := TRUE;
   END_IF;
END_REGION

REGION Network 8
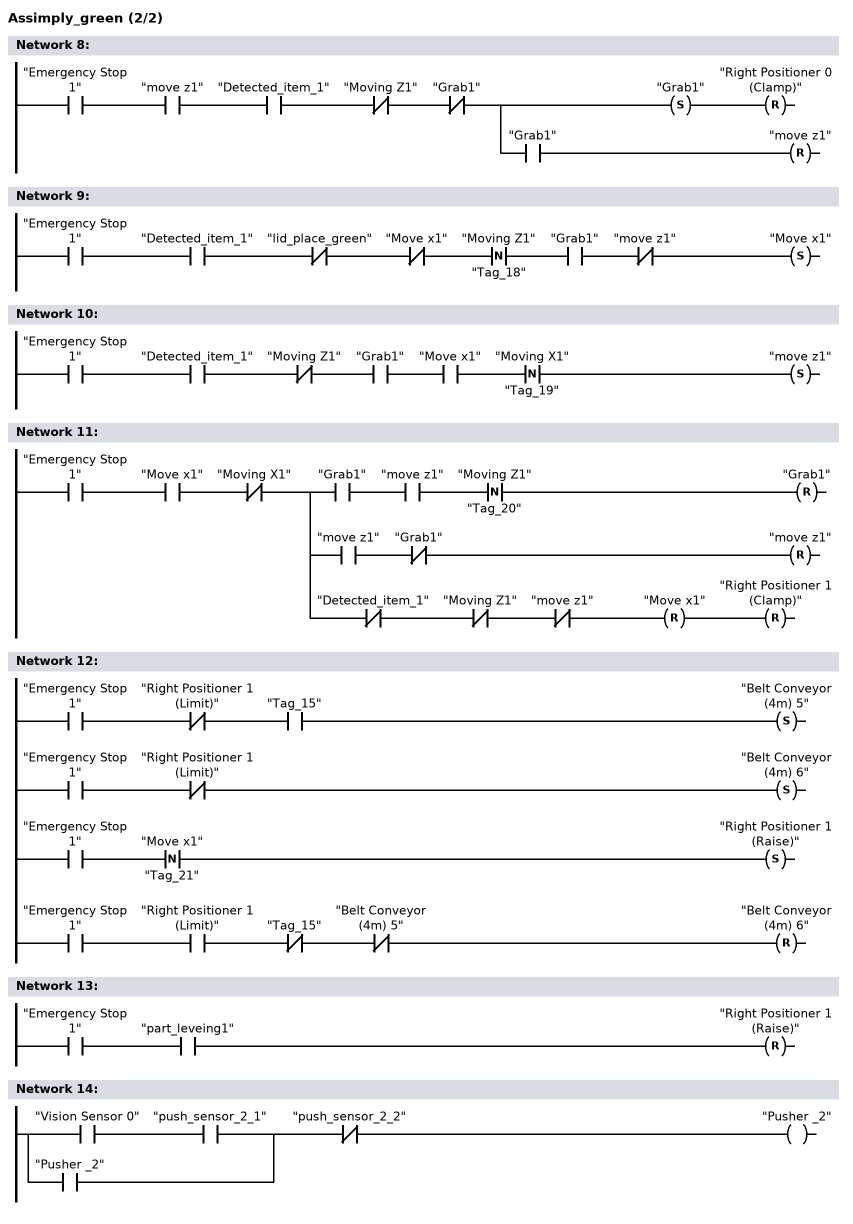
   RUNG wire#powerrail
      Contact( "Emergency Stop 1" )
      Contact( "move z1" )
      Contact( "Detected_item_1" )
      I_Contact( "Moving Z1" )
      I_Contact( "Grab1" )
      wire#w1
      S_Coil( "Grab1" )
      R_Coil( "Right Positioner 0 (Clamp)" )
   END_RUNG
   RUNG wire#w1
      Contact( "Grab1" )
      R_Coil( "move z1" )
   END_RUNG
   // the same network as SCL:
   #_w1 := "Emergency Stop 1" AND "move z1" AND "Detected_item_1" AND NOT "Moving Z1" AND NOT "Grab1";
   IF #_w1 THEN
       "Grab1" := TRUE;
       "Right Positioner 0 (Clamp)" := FALSE;
   END_IF;
   IF #_w1 AND "Grab1" THEN "move z1" := FALSE; END_IF;
END_REGION

REGION Network 9
   RUNG wire#powerrail
      Contact( "Emergency Stop 1" )
      Contact( "Detected_item_1" )
      I_Contact( "lid_place_green" )
      I_Contact( "Move x1" )
      N_Contact(operand := "Moving Z1", bit := "Tag_18")
      Contact( "Grab1" )
      I_Contact( "move z1" )
      S_Coil( "Move x1" )
   END_RUNG
   // the same network as SCL:
   #_w1 := "Emergency Stop 1" AND "Detected_item_1" AND NOT "lid_place_green" AND NOT "Move x1" AND NOT "Moving Z1" AND "Tag_18";   // falling edge of "Moving Z1"
   "Tag_18" := "Moving Z1";
   IF #_w1 AND "Grab1" AND NOT "move z1" THEN "Move x1" := TRUE; END_IF;
END_REGION

REGION Network 10
   RUNG wire#powerrail
      Contact( "Emergency Stop 1" )
      Contact( "Detected_item_1" )
      I_Contact( "Moving Z1" )
      Contact( "Grab1" )
      Contact( "Move x1" )
      N_Contact(operand := "Moving X1", bit := "Tag_19")
      S_Coil( "move z1" )
   END_RUNG
   // the same network as SCL:
   #_w1 := "Emergency Stop 1" AND "Detected_item_1" AND NOT "Moving Z1" AND "Grab1" AND "Move x1" AND NOT "Moving X1" AND "Tag_19";   // falling edge of "Moving X1"
   "Tag_19" := "Moving X1";
   IF #_w1 THEN "move z1" := TRUE; END_IF;
END_REGION

REGION Network 11
   RUNG wire#powerrail
      Contact( "Emergency Stop 1" )
      Contact( "Move x1" )
      I_Contact( "Moving X1" )
      wire#w1
      Contact( "Grab1" )
      Contact( "move z1" )
      N_Contact(operand := "Moving Z1", bit := "Tag_20")
      R_Coil( "Grab1" )
   END_RUNG
   RUNG wire#w1
      Contact( "move z1" )
      I_Contact( "Grab1" )
      R_Coil( "move z1" )
   END_RUNG
   RUNG wire#w1
      I_Contact( "Detected_item_1" )
      I_Contact( "Moving Z1" )
      I_Contact( "move z1" )
      R_Coil( "Move x1" )
      R_Coil( "Right Positioner 1 (Clamp)" )
   END_RUNG
   // the same network as SCL:
   #_w1 := "Emergency Stop 1" AND "Move x1" AND NOT "Moving X1";
   #_w2 := #_w1 AND "Grab1" AND "move z1" AND NOT "Moving Z1" AND "Tag_20";   // falling edge of "Moving Z1"
   "Tag_20" := "Moving Z1";
   IF #_w2 THEN "Grab1" := FALSE; END_IF;
   IF #_w1 AND "move z1" AND NOT "Grab1" THEN "move z1" := FALSE; END_IF;
   IF #_w1 AND NOT "Detected_item_1" AND NOT "Moving Z1" AND NOT "move z1" THEN
       "Move x1" := FALSE;
       "Right Positioner 1 (Clamp)" := FALSE;
   END_IF;
END_REGION

REGION Network 12
   RUNG wire#powerrail
      Contact( "Emergency Stop 1" )
      I_Contact( "Right Positioner 1 (Limit)" )
      Contact( "Tag_15" )
      S_Coil( "Belt Conveyor (4m) 5" )
   END_RUNG
   RUNG wire#powerrail
      Contact( "Emergency Stop 1" )
      I_Contact( "Right Positioner 1 (Limit)" )
      S_Coil( "Belt Conveyor (4m) 6" )
   END_RUNG
   RUNG wire#powerrail
      Contact( "Emergency Stop 1" )
      N_Contact(operand := "Move x1", bit := "Tag_21")
      S_Coil( "Right Positioner 1 (Raise)" )
   END_RUNG
   RUNG wire#powerrail
      Contact( "Emergency Stop 1" )
      Contact( "Right Positioner 1 (Limit)" )
      I_Contact( "Tag_15" )
      I_Contact( "Belt Conveyor (4m) 5" )
      R_Coil( "Belt Conveyor (4m) 6" )
   END_RUNG
   // the same network as SCL:
   IF "Emergency Stop 1" AND NOT "Right Positioner 1 (Limit)" AND "Tag_15" THEN
       "Belt Conveyor (4m) 5" := TRUE;
   END_IF;
   IF "Emergency Stop 1" AND NOT "Right Positioner 1 (Limit)" THEN "Belt Conveyor (4m) 6" := TRUE; END_IF;
   #_w1 := "Emergency Stop 1" AND NOT "Move x1" AND "Tag_21";   // falling edge of "Move x1"
   "Tag_21" := "Move x1";
   IF #_w1 THEN "Right Positioner 1 (Raise)" := TRUE; END_IF;
   IF "Emergency Stop 1" AND "Right Positioner 1 (Limit)" AND NOT "Tag_15" AND NOT "Belt Conveyor (4m) 5" THEN
       "Belt Conveyor (4m) 6" := FALSE;
   END_IF;
END_REGION

REGION Network 13
   RUNG wire#powerrail
      Contact( "Emergency Stop 1" )
      Contact( "part_leveing1" )
      R_Coil( "Right Positioner 1 (Raise)" )
   END_RUNG
   // the same network as SCL:
   IF "Emergency Stop 1" AND "part_leveing1" THEN "Right Positioner 1 (Raise)" := FALSE; END_IF;
END_REGION

REGION Network 14
   RUNG wire#powerrail
      Contact( "Vision Sensor 0" )
      Contact( "push_sensor_2_1" )
      wire#w1
      I_Contact( "push_sensor_2_2" )
      Coil( "Pusher _2" )
   END_RUNG
   RUNG wire#powerrail
      Contact( "Pusher _2" )
   END_RUNG wire#w1
   // the same network as SCL:
   "Pusher _2" := (("Vision Sensor 0" AND "push_sensor_2_1") OR "Pusher _2") AND NOT "push_sensor_2_2";
END_REGION
END_FUNCTION

FUNCTION "assimply_blue" : Void   // FC8, LAD
{ S7_Optimized_Access := 'TRUE' }
VERSION : 0.1
   VAR_TEMP   // added for the SCL form of the ladder/FBD networks
      _w1 : Bool;
      _w2 : Bool;
   END_VAR
BEGIN

REGION Network 1
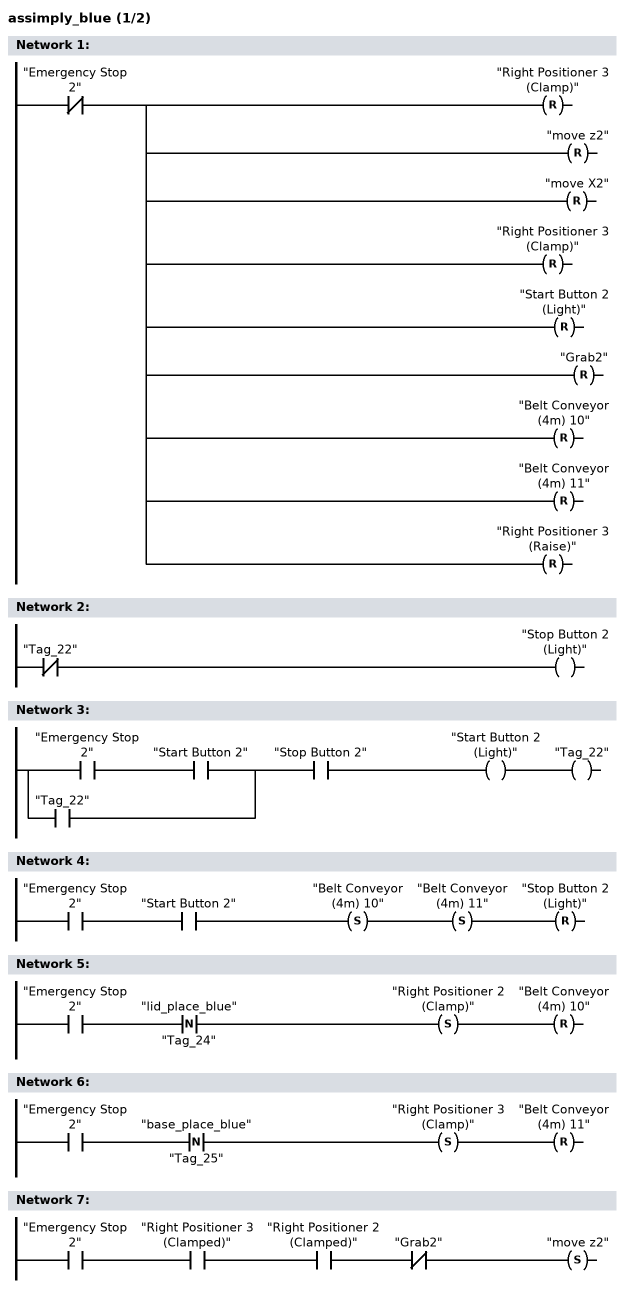
   RUNG wire#powerrail
      I_Contact( "Emergency Stop 2" )
      wire#w1
      R_Coil( "Right Positioner 3 (Clamp)" )
   END_RUNG
   RUNG wire#w1
      R_Coil( "move z2" )
   END_RUNG
   RUNG wire#w1
      R_Coil( "move X2" )
   END_RUNG
   RUNG wire#w1
      R_Coil( "Right Positioner 3 (Clamp)" )
   END_RUNG
   RUNG wire#w1
      R_Coil( "Start Button 2 (Light)" )
   END_RUNG
   RUNG wire#w1
      R_Coil( "Grab2" )
   END_RUNG
   RUNG wire#w1
      R_Coil( "Belt Conveyor (4m) 10" )
   END_RUNG
   RUNG wire#w1
      R_Coil( "Belt Conveyor (4m) 11" )
   END_RUNG
   RUNG wire#w1
      R_Coil( "Right Positioner 3 (Raise)" )
   END_RUNG
   // the same network as SCL:
   IF NOT "Emergency Stop 2" THEN
       "Right Positioner 3 (Clamp)" := FALSE;
       "move z2" := FALSE;
       "move X2" := FALSE;
       "Right Positioner 3 (Clamp)" := FALSE;
       "Start Button 2 (Light)" := FALSE;
       "Grab2" := FALSE;
       "Belt Conveyor (4m) 10" := FALSE;
       "Belt Conveyor (4m) 11" := FALSE;
       "Right Positioner 3 (Raise)" := FALSE;
   END_IF;
END_REGION

REGION Network 2
   RUNG wire#powerrail
      I_Contact( "Tag_22" )
      Coil( "Stop Button 2 (Light)" )
   END_RUNG
   // the same network as SCL:
   "Stop Button 2 (Light)" := NOT "Tag_22";
END_REGION

REGION Network 3
   RUNG wire#powerrail
      Contact( "Emergency Stop 2" )
      Contact( "Start Button 2" )
      wire#w1
      Contact( "Stop Button 2" )
      Coil( "Start Button 2 (Light)" )
      Coil( "Tag_22" )
   END_RUNG
   RUNG wire#powerrail
      Contact( "Tag_22" )
   END_RUNG wire#w1
   // the same network as SCL:
   "Start Button 2 (Light)" := (("Emergency Stop 2" AND "Start Button 2") OR "Tag_22") AND "Stop Button 2";
   "Tag_22" := "Start Button 2 (Light)";
END_REGION

REGION Network 4
   RUNG wire#powerrail
      Contact( "Emergency Stop 2" )
      Contact( "Start Button 2" )
      S_Coil( "Belt Conveyor (4m) 10" )
      S_Coil( "Belt Conveyor (4m) 11" )
      R_Coil( "Stop Button 2 (Light)" )
   END_RUNG
   // the same network as SCL:
   IF "Emergency Stop 2" AND "Start Button 2" THEN
       "Belt Conveyor (4m) 10" := TRUE;
       "Belt Conveyor (4m) 11" := TRUE;
       "Stop Button 2 (Light)" := FALSE;
   END_IF;
END_REGION

REGION Network 5
   RUNG wire#powerrail
      Contact( "Emergency Stop 2" )
      N_Contact(operand := "lid_place_blue", bit := "Tag_24")
      S_Coil( "Right Positioner 2 (Clamp)" )
      R_Coil( "Belt Conveyor (4m) 10" )
   END_RUNG
   // the same network as SCL:
   #_w1 := "Emergency Stop 2" AND NOT "lid_place_blue" AND "Tag_24";   // falling edge of "lid_place_blue"
   "Tag_24" := "lid_place_blue";
   IF #_w1 THEN
       "Right Positioner 2 (Clamp)" := TRUE;
       "Belt Conveyor (4m) 10" := FALSE;
   END_IF;
END_REGION

REGION Network 6
   RUNG wire#powerrail
      Contact( "Emergency Stop 2" )
      N_Contact(operand := "base_place_blue", bit := "Tag_25")
      S_Coil( "Right Positioner 3 (Clamp)" )
      R_Coil( "Belt Conveyor (4m) 11" )
   END_RUNG
   // the same network as SCL:
   #_w1 := "Emergency Stop 2" AND NOT "base_place_blue" AND "Tag_25";   // falling edge of "base_place_blue"
   "Tag_25" := "base_place_blue";
   IF #_w1 THEN
       "Right Positioner 3 (Clamp)" := TRUE;
       "Belt Conveyor (4m) 11" := FALSE;
   END_IF;
END_REGION

REGION Network 7
   RUNG wire#powerrail
      Contact( "Emergency Stop 2" )
      Contact( "Right Positioner 3 (Clamped)" )
      Contact( "Right Positioner 2 (Clamped)" )
      I_Contact( "Grab2" )
      S_Coil( "move z2" )
   END_RUNG
   // the same network as SCL:
   IF "Emergency Stop 2" AND "Right Positioner 3 (Clamped)" AND "Right Positioner 2 (Clamped)" AND NOT "Grab2" THEN
       "move z2" := TRUE;
   END_IF;
END_REGION

REGION Network 8
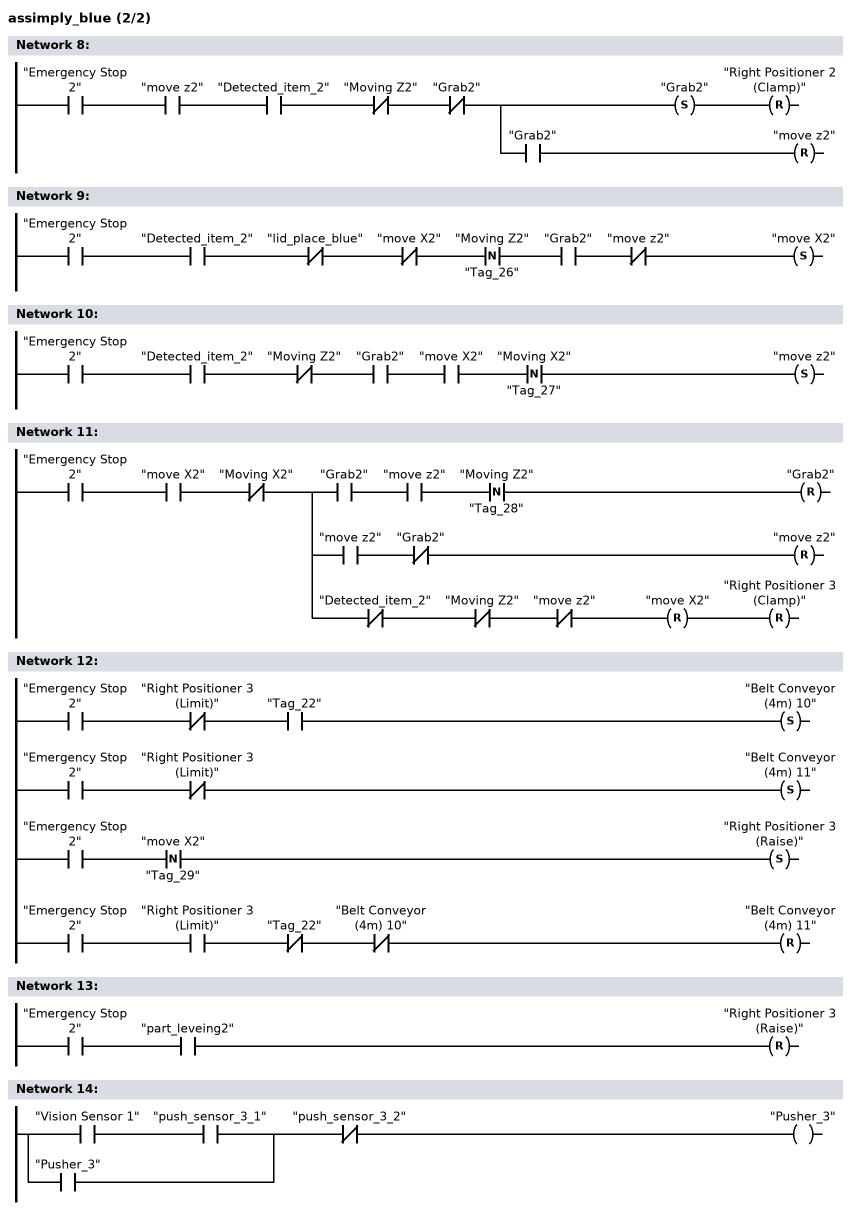
   RUNG wire#powerrail
      Contact( "Emergency Stop 2" )
      Contact( "move z2" )
      Contact( "Detected_item_2" )
      I_Contact( "Moving Z2" )
      I_Contact( "Grab2" )
      wire#w1
      S_Coil( "Grab2" )
      R_Coil( "Right Positioner 2 (Clamp)" )
   END_RUNG
   RUNG wire#w1
      Contact( "Grab2" )
      R_Coil( "move z2" )
   END_RUNG
   // the same network as SCL:
   #_w1 := "Emergency Stop 2" AND "move z2" AND "Detected_item_2" AND NOT "Moving Z2" AND NOT "Grab2";
   IF #_w1 THEN
       "Grab2" := TRUE;
       "Right Positioner 2 (Clamp)" := FALSE;
   END_IF;
   IF #_w1 AND "Grab2" THEN "move z2" := FALSE; END_IF;
END_REGION

REGION Network 9
   RUNG wire#powerrail
      Contact( "Emergency Stop 2" )
      Contact( "Detected_item_2" )
      I_Contact( "lid_place_blue" )
      I_Contact( "move X2" )
      N_Contact(operand := "Moving Z2", bit := "Tag_26")
      Contact( "Grab2" )
      I_Contact( "move z2" )
      S_Coil( "move X2" )
   END_RUNG
   // the same network as SCL:
   #_w1 := "Emergency Stop 2" AND "Detected_item_2" AND NOT "lid_place_blue" AND NOT "move X2" AND NOT "Moving Z2" AND "Tag_26";   // falling edge of "Moving Z2"
   "Tag_26" := "Moving Z2";
   IF #_w1 AND "Grab2" AND NOT "move z2" THEN "move X2" := TRUE; END_IF;
END_REGION

REGION Network 10
   RUNG wire#powerrail
      Contact( "Emergency Stop 2" )
      Contact( "Detected_item_2" )
      I_Contact( "Moving Z2" )
      Contact( "Grab2" )
      Contact( "move X2" )
      N_Contact(operand := "Moving X2", bit := "Tag_27")
      S_Coil( "move z2" )
   END_RUNG
   // the same network as SCL:
   #_w1 := "Emergency Stop 2" AND "Detected_item_2" AND NOT "Moving Z2" AND "Grab2" AND "move X2" AND NOT "Moving X2" AND "Tag_27";   // falling edge of "Moving X2"
   "Tag_27" := "Moving X2";
   IF #_w1 THEN "move z2" := TRUE; END_IF;
END_REGION

REGION Network 11
   RUNG wire#powerrail
      Contact( "Emergency Stop 2" )
      Contact( "move X2" )
      I_Contact( "Moving X2" )
      wire#w1
      Contact( "Grab2" )
      Contact( "move z2" )
      N_Contact(operand := "Moving Z2", bit := "Tag_28")
      R_Coil( "Grab2" )
   END_RUNG
   RUNG wire#w1
      Contact( "move z2" )
      I_Contact( "Grab2" )
      R_Coil( "move z2" )
   END_RUNG
   RUNG wire#w1
      I_Contact( "Detected_item_2" )
      I_Contact( "Moving Z2" )
      I_Contact( "move z2" )
      R_Coil( "move X2" )
      R_Coil( "Right Positioner 3 (Clamp)" )
   END_RUNG
   // the same network as SCL:
   #_w1 := "Emergency Stop 2" AND "move X2" AND NOT "Moving X2";
   #_w2 := #_w1 AND "Grab2" AND "move z2" AND NOT "Moving Z2" AND "Tag_28";   // falling edge of "Moving Z2"
   "Tag_28" := "Moving Z2";
   IF #_w2 THEN "Grab2" := FALSE; END_IF;
   IF #_w1 AND "move z2" AND NOT "Grab2" THEN "move z2" := FALSE; END_IF;
   IF #_w1 AND NOT "Detected_item_2" AND NOT "Moving Z2" AND NOT "move z2" THEN
       "move X2" := FALSE;
       "Right Positioner 3 (Clamp)" := FALSE;
   END_IF;
END_REGION

REGION Network 12
   RUNG wire#powerrail
      Contact( "Emergency Stop 2" )
      I_Contact( "Right Positioner 3 (Limit)" )
      Contact( "Tag_22" )
      S_Coil( "Belt Conveyor (4m) 10" )
   END_RUNG
   RUNG wire#powerrail
      Contact( "Emergency Stop 2" )
      I_Contact( "Right Positioner 3 (Limit)" )
      S_Coil( "Belt Conveyor (4m) 11" )
   END_RUNG
   RUNG wire#powerrail
      Contact( "Emergency Stop 2" )
      N_Contact(operand := "move X2", bit := "Tag_29")
      S_Coil( "Right Positioner 3 (Raise)" )
   END_RUNG
   RUNG wire#powerrail
      Contact( "Emergency Stop 2" )
      Contact( "Right Positioner 3 (Limit)" )
      I_Contact( "Tag_22" )
      I_Contact( "Belt Conveyor (4m) 10" )
      R_Coil( "Belt Conveyor (4m) 11" )
   END_RUNG
   // the same network as SCL:
   IF "Emergency Stop 2" AND NOT "Right Positioner 3 (Limit)" AND "Tag_22" THEN
       "Belt Conveyor (4m) 10" := TRUE;
   END_IF;
   IF "Emergency Stop 2" AND NOT "Right Positioner 3 (Limit)" THEN "Belt Conveyor (4m) 11" := TRUE; END_IF;
   #_w1 := "Emergency Stop 2" AND NOT "move X2" AND "Tag_29";   // falling edge of "move X2"
   "Tag_29" := "move X2";
   IF #_w1 THEN "Right Positioner 3 (Raise)" := TRUE; END_IF;
   IF "Emergency Stop 2" AND "Right Positioner 3 (Limit)" AND NOT "Tag_22" AND NOT "Belt Conveyor (4m) 10" THEN
       "Belt Conveyor (4m) 11" := FALSE;
   END_IF;
END_REGION

REGION Network 13
   RUNG wire#powerrail
      Contact( "Emergency Stop 2" )
      Contact( "part_leveing2" )
      R_Coil( "Right Positioner 3 (Raise)" )
   END_RUNG
   // the same network as SCL:
   IF "Emergency Stop 2" AND "part_leveing2" THEN "Right Positioner 3 (Raise)" := FALSE; END_IF;
END_REGION

REGION Network 14
   RUNG wire#powerrail
      Contact( "Vision Sensor 1" )
      Contact( "push_sensor_3_1" )
      wire#w1
      I_Contact( "push_sensor_3_2" )
      Coil( "Pusher_3" )
   END_RUNG
   RUNG wire#powerrail
      Contact( "Pusher_3" )
   END_RUNG wire#w1
   // the same network as SCL:
   "Pusher_3" := (("Vision Sensor 1" AND "push_sensor_3_1") OR "Pusher_3") AND NOT "push_sensor_3_2";
END_REGION
END_FUNCTION

FUNCTION "COUNTER_FN" : Void   // FC9, LAD
{ S7_Optimized_Access := 'TRUE' }
VERSION : 0.1
   VAR_TEMP   // added for the SCL form of the ladder/FBD networks
      _w1 : Bool;
   END_VAR
BEGIN

REGION Network 1
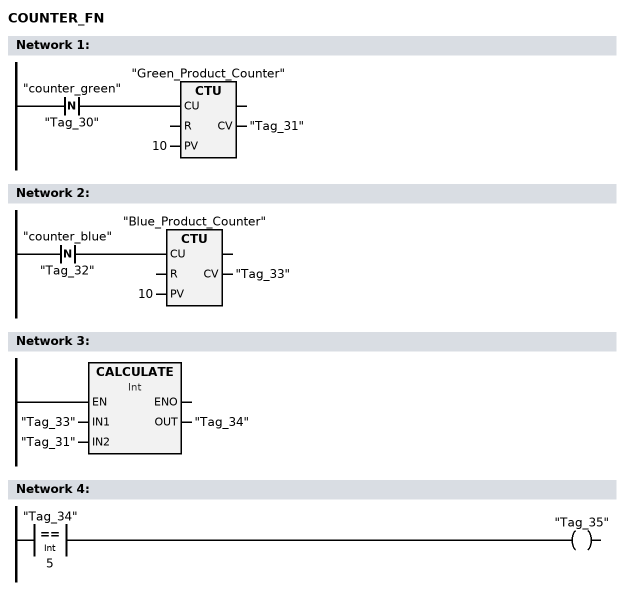
   #_w1 := NOT "counter_green" AND "Tag_30";   // falling edge of "counter_green"
   "Tag_30" := "counter_green";
   "Green_Product_Counter".CTU(CU := #_w1, PV := 10, CV => "Tag_31");
END_REGION

REGION Network 2
   #_w1 := NOT "counter_blue" AND "Tag_32";   // falling edge of "counter_blue"
   "Tag_32" := "counter_blue";
   "Blue_Product_Counter".CTU(CU := #_w1, PV := 10, CV => "Tag_33");
END_REGION

REGION Network 3
   RUNG wire#powerrail
      { S7_Templates := "SrcType := Int"; S7_Expression := "(IN1+IN2)" } Calculate(in1 := "Tag_33", in2 := "Tag_31", out => "Tag_34")
   END_RUNG
   // the same network as SCL:
   "Tag_34" := ("Tag_33"+"Tag_31");
END_REGION

REGION Network 4
   RUNG wire#powerrail
      { S7_Templates := "SrcType := Int" } EQ_Contact(in1 := "Tag_34", in2 := 5)
      Coil( "Tag_35" )
   END_RUNG
   // the same network as SCL:
   "Tag_35" := "Tag_34" = 5;
END_REGION
END_FUNCTION

FUNCTION "MHJ-PLC-Lab-Function-S71200" : Void   // FC9000, SCL
{ S7_Optimized_Access := 'TRUE' }
VERSION : 0.1
   VAR_TEMP
      rdTimeReturn : Int;
      outputTime : DTL;
      SyncVal : Byte;
      forVal : Int;
      forVal_2 : Int;
      Value : Byte;
   END_VAR
   VAR CONSTANT
      CompVal : Byte := 16#34;
      Value_01 : Byte := 16#11;
      Value_01_DW : DWord := 16#A165_D992;
      Value_02_DW : DWord := 16#58BE_4401;
   END_VAR
BEGIN

   #Value:=PEEK(area := 16#82,
        dbNumber := 0,
        byteOffset := 511);
   #Value := #Value + 1;

   POKE(area := 16#82,
        dbNumber := 0,
        byteOffset := 511,
        value := #Value);

   POKE(area:=16#81,
        dbNumber:=0,
        byteOffset:=1016,
        value:=#Value_01_DW);
   POKE(area := 16#81,
        dbNumber := 0,
        byteOffset := 1020,
        value := #Value_02_DW);

   POKE(area := 16#81,
        dbNumber := 0,
        byteOffset := 511,
        value := B#16#00);

   FOR #forVal := 0 TO 120 DO
       FOR #forVal_2:=0 TO 10 DO
           #rdTimeReturn:=RD_SYS_T(#outputTime);
           #rdTimeReturn := WR_SYS_T(#outputTime);
           #rdTimeReturn := RD_SYS_T(#outputTime);
           #rdTimeReturn := WR_SYS_T(#outputTime);
       END_FOR;
       #SyncVal:= PEEK(area := 16#81,
                      dbNumber := 0,
                      byteOffset := 511);
       IF #SyncVal = #CompVal THEN
          GOTO M_1;
       END_IF;
   END_FOR;
   RETURN;

   M_1:
   POKE(area := 16#81,
        dbNumber := 0,
        byteOffset := 511,
        value := B#16#0);
END_FUNCTION

ORGANIZATION_BLOCK "Main"   // OB1, LAD, ProgramCycle
TITLE = "Main Program Sweep (Cycle)"
{ S7_Optimized_Access := 'TRUE' }
VERSION : 0.1
   VAR_INPUT
      Initial_Call : Bool;   // Initial call of this OB
      Remanence : Bool;   // =True, if remanent data are available
   END_VAR
BEGIN

REGION Network 1: Konnektierungsbaustein für PLC-Lab
   // Im Netzwerk 1 wird der Konnektierungsbaustein für PLC-Lab aufgerufen.
   // Dieser Aufruf darf nicht entfernt werden!
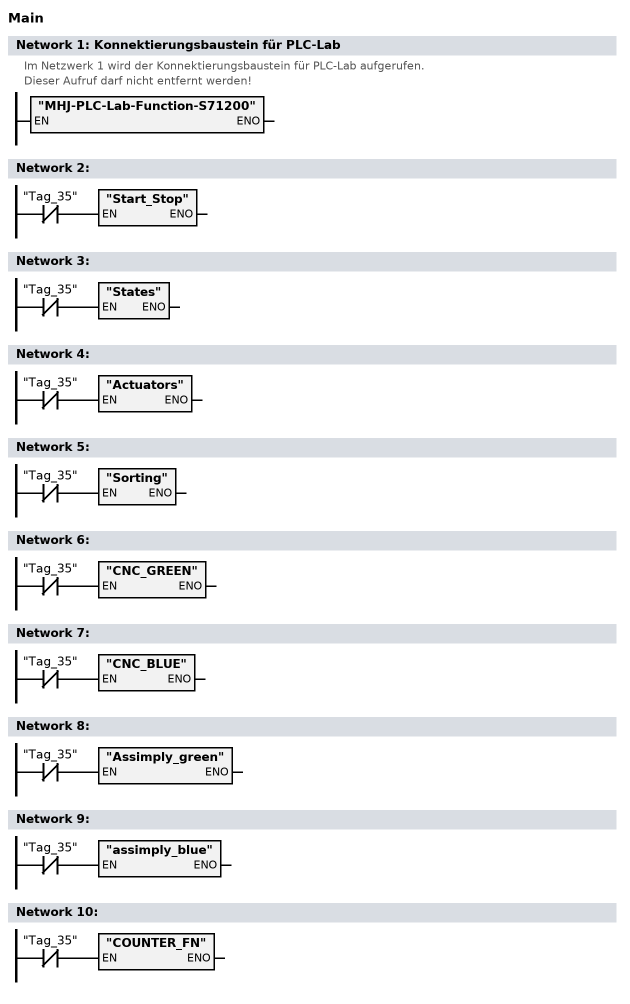
   RUNG wire#powerrail
      "MHJ-PLC-Lab-Function-S71200"()
   END_RUNG
   // the same network as SCL:
   "MHJ-PLC-Lab-Function-S71200"();
END_REGION

REGION Network 2
   RUNG wire#powerrail
      I_Contact( "Tag_35" )
      "Start_Stop"()
   END_RUNG
   // the same network as SCL:
   IF NOT "Tag_35" THEN "Start_Stop"(); END_IF;
END_REGION

REGION Network 3
   RUNG wire#powerrail
      I_Contact( "Tag_35" )
      "States"()
   END_RUNG
   // the same network as SCL:
   IF NOT "Tag_35" THEN "States"(); END_IF;
END_REGION

REGION Network 4
   RUNG wire#powerrail
      I_Contact( "Tag_35" )
      "Actuators"()
   END_RUNG
   // the same network as SCL:
   IF NOT "Tag_35" THEN "Actuators"(); END_IF;
END_REGION

REGION Network 5
   RUNG wire#powerrail
      I_Contact( "Tag_35" )
      "Sorting"()
   END_RUNG
   // the same network as SCL:
   IF NOT "Tag_35" THEN "Sorting"(); END_IF;
END_REGION

REGION Network 6
   RUNG wire#powerrail
      I_Contact( "Tag_35" )
      "CNC_GREEN"()
   END_RUNG
   // the same network as SCL:
   IF NOT "Tag_35" THEN "CNC_GREEN"(); END_IF;
END_REGION

REGION Network 7
   RUNG wire#powerrail
      I_Contact( "Tag_35" )
      "CNC_BLUE"()
   END_RUNG
   // the same network as SCL:
   IF NOT "Tag_35" THEN "CNC_BLUE"(); END_IF;
END_REGION

REGION Network 8
   RUNG wire#powerrail
      I_Contact( "Tag_35" )
      "Assimply_green"()
   END_RUNG
   // the same network as SCL:
   IF NOT "Tag_35" THEN "Assimply_green"(); END_IF;
END_REGION

REGION Network 9
   RUNG wire#powerrail
      I_Contact( "Tag_35" )
      "assimply_blue"()
   END_RUNG
   // the same network as SCL:
   IF NOT "Tag_35" THEN "assimply_blue"(); END_IF;
END_REGION

REGION Network 10
   RUNG wire#powerrail
      I_Contact( "Tag_35" )
      "COUNTER_FN"()
   END_RUNG
   // the same network as SCL:
   IF NOT "Tag_35" THEN "COUNTER_FN"(); END_IF;
END_REGION
END_ORGANIZATION_BLOCK

ORGANIZATION_BLOCK "Startup"   // OB100, LAD, Startup
TITLE = "Complete Restart"
{ S7_Optimized_Access := 'TRUE' }
VERSION : 0.1
   VAR_INPUT
      LostRetentive : Bool;   // True if retentive data are lost
      LostRTC : Bool;   // True if date and time are lost
   END_VAR
BEGIN

REGION Network 1
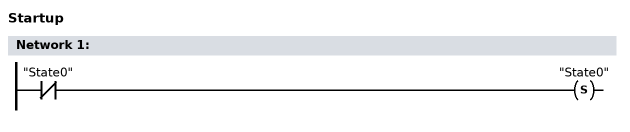
   RUNG wire#powerrail
      I_Contact( "State0" )
      S_Coil( "State0" )
   END_RUNG
   // the same network as SCL:
   IF NOT "State0" THEN "State0" := TRUE; END_IF;
END_REGION
END_ORGANIZATION_BLOCK

(* ===== HMI "HMI_RT_1" =====
system functions are stored by id; their names below are inferred from use
connection "HMI_Connection_1": ETHERNET, S7_1200_OMS

HMI tags "Default tag table"
   "start button0" : Bool = PLC "Start Button 0" AT %I0.5, 1 s
   "Start buttono light" : Bool = PLC "Start Button 0 (Light)" AT %Q0.5, 1 s
   "stop button0" : Bool = PLC "Stop Button 0" AT %I0.6, 1 s
   "stop button 0 light" : Bool = PLC "Stop Button 0 (Light)" AT %Q0.6, 1 s
   "green on" : Bool = PLC "Machining green(Start)" AT %Q2.1, 1 s
   "Blue on" : Bool = PLC "Machining blue 0 (Start)" AT %Q6.6, 1 s
   "start button1" : Bool = PLC "Start Button 1" AT %I2.2, 1 s
   "start button2" : Bool = PLC "Start Button 2" AT %I2.5, 1 s
   "stop button1" : Bool = PLC "Stop Button 1" AT %I2.3, 1 s
   "stop button2" : Bool = PLC "Stop Button 2" AT %I2.6, 1 s
   "Start button1 light" : Bool = PLC "Start Button 1 (Light)" AT %Q2.7, 1 s
   "Start button2 light" : Bool = PLC "Start Button 2 (Light)" AT %Q3.1, 1 s
   "stop button 1 light" : Bool = PLC "Stop Button 1 (Light)" AT %Q3.0, 1 s
   "stop button 2 light" : Bool = PLC "Stop Button 2 (Light)" AT %Q3.2, 1 s
   "tag31" : Int = PLC Tag_31 AT %MW400, 1 s
   "tag33" : Int = PLC Tag_33 AT %MW500, 1 s
   "tag35" : Int = PLC Tag_34 AT %MW600, 1 s

text list "Busy or not": 0 'not busy'; 1 'busy'

Template "ScrNav" 800x409
   Button "Template_Button_1" at 19,351 size 141x40; TextOff 'Home'
      on Click: ActivateScreen("Home", 0)
   Button "Template_Button_2" at 190,350 size 125x43; TextOff 'Green CNC'
      on Click: ActivateScreen("Green CNC", 0)
   Button "Template_Button_3" at 341,350 size 121x42; TextOff 'Blue CNC'
      on Click: ActivateScreen("Blue CNC", 0)

screen "Home" 800x409, template "ScrNav"
   TextField "Text field_1" at 340,13 size 139x23; Text 'Home screen...'
   Button "Button_1" at 49,65 size 111x51; TextOff 'Start'
      on Press: function_b14e0dd5("start button0", 0)
      Appearance <- "Start buttono light"
   Button "Button_2" at 48,141 size 110x48; TextOff 'Stop'
      on Press: function_b14e0dd5("stop button0", 0)
      Appearance <- "stop button 0 light"
   Circle "Circle_1" at 268,65 size 48x48
      Appearance <- "Start buttono light"
   Circle "Circle_2" at 268,141 size 48x48
      Appearance <- "stop button 0 light"
   TextField "Text field_2" at 484,73 size 138x27; Text 'Green CNC...'
   Circle "Circle_4" at 667,64 size 48x48
      Appearance <- "green on"
   TextField "Text field_3" at 493,144 size 123x27; Text 'Blue CNC...'
   Circle "Circle_5" at 667,133 size 48x48
      Appearance <- "Blue on"
   Clock "Clock_1" at 674,289 size 120x120
   IOField "I/O field_1" at 426,220 size 110x53; FormatPattern s99999
      ProcessValue <- "tag35"
   TextField "Text field_4" at 208,234 size 204x29; Text 'Total products:...'

screen "Green CNC" 800x409, template "ScrNav"
   TextField "Text field_1" at 331,12 size 185x23; Text 'Green CNC screen...'
   TextField "Text field_2" at 421,102 size 182x27; Text 'State of CNC:...'
   SymbolicIOField "Symbolic I/O field_1" at 591,84 size 170x54; TextOn '1'; TextOff '0'; TextList "Busy or not"
      ProcessValue <- "green on"
   IOField "I/O field_1" at 272,223 size 102x56; FormatPattern s99999
      ProcessValue <- "tag31"
   TextField "Text field_3" at 30,237 size 232x27; Text 'Number of product:...'
   Button "Button_1" at 49,65 size 111x51; TextOff 'Start'
      on Press: function_b14e0dd5("start button1", 0)
      Appearance <- "Start button1 light"
   Button "Button_2" at 48,141 size 110x48; TextOff 'Stop'
      on Press: function_b14e0dd5("stop button1", 0)
      Appearance <- "stop button 1 light"
   Circle "Circle_2" at 268,65 size 48x48
      Appearance <- "Start button1 light"
   Circle "Circle_3" at 268,141 size 48x48
      Appearance <- "stop button 1 light"

screen "Blue CNC" 800x409, template "ScrNav"
   TextField "Text field_1" at 331,12 size 171x23; Text 'Blue CNC screen...'
   TextField "Text field_2" at 421,102 size 182x27; Text 'State of CNC:...'
   SymbolicIOField "Symbolic I/O field_1" at 591,84 size 170x54; TextOn '1'; TextOff '0'; TextList "Busy or not"
      ProcessValue <- "tag31"
   IOField "I/O field_1" at 272,223 size 102x56; FormatPattern s99999
      ProcessValue <- "tag33"
   TextField "Text field_3" at 30,237 size 232x27; Text 'Number of product:...'
   Button "Button_1" at 49,65 size 111x51; TextOff 'Start'
      on Press: function_b14e0dd5("start button2", 0)
      Appearance <- "Start button2 light"
   Button "Button_2" at 48,141 size 110x48; TextOff 'Stop'
      on Press: function_b14e0dd5("stop button2", 0)
      Appearance <- "stop button 2 light"
   Circle "Circle_2" at 268,65 size 48x48
      Appearance <- "Start button2 light"
   Circle "Circle_3" at 268,141 size 48x48
      Appearance <- "stop button 2 light"
*)